Fanuc KAREL source: rsi_position.kl

PROGRAM rsiposition

%COMMENT = 'rsiposition v1'
%NOLOCKGROUP
%NOBUSYLAMP

VAR
	rf_ :FILE
	STATUS: INTEGER
	current_pos: XYZWPR

BEGIN

	current_pos = CURPOS(0,0)
	OPEN FILE rf_ ('RW', 'RD:RESPONSE.HTM')
	STATUS = IO_STATUS(rf_)
	IF (STATUS <> 0) THEN
		WRITE rf_ ( '{"result":"failed", "program":"rsiposition", "reason":',STATUS,'}')
	ELSE
		WRITE rf_ ( '{"x":', current_pos.x,
					', "y":', current_pos.y,
					', "z":', current_pos.z,
					', "w":', current_pos.w,
					', "p":', current_pos.p,
					', "r":', current_pos.r,
					'}')
	ENDIF
	CLOSE FILE rf_
END rsiposition
